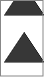
VISUALIZATION ValveDiagonal  // 44x77
VAR_IN_OUT
	valve_toggleColor : BOOL;
	valve_tapVariable : BOOL;
END_VAR
    Polygon (4,15) (24,-15) (44,15) (33,15) (19,15), colour toggle: valve_toggleColor
        tap valve_tapVariable
    Polygon (4,62) (24,32) (44,62) (33,62) (19,62), colour toggle: valve_toggleColor
        tap valve_tapVariable
END_VISUALIZATION

(* stored: Version 1.1.0.1, ProductVersion 3.1.4024.9
   Visu ValveDiagonal: Id {f18b39c6-66da-47e3-9fba-089bb84f82f4} *)
